FUNCTION_BLOCK AxisMovementController
VAR_INPUT
	tolerance: UINT;
	desiredSpeed: INT;
	currentPosition : UINT;
	requiredPosition : UINT;
END_VAR
VAR_OUTPUT
	AxisMinus : BOOL;
	AxisPlus: BOOL;
	Control: INT;
	SpeedPWM:INT;
	InPosition:BOOL;
END_VAR
VAR
END_VAR

IF  AboutEqual(
	uiActual:= currentPosition,
	uiRequiered:= requiredPosition,
	uiTolerance:= tolerance
)
 THEN
	AxisMinus := FALSE;
	AxisPlus := FALSE;
	Control := 0;
	SpeedPWM := 0;
	InPosition := TRUE;
ELSIF currentPosition > requiredPosition AND NOT InPosition THEN
	AxisMinus := TRUE;
	AxisPlus := FALSE;
	Control:= 32;
	SpeedPWM := desiredSpeed;
	InPosition := FALSE;
ELSIF currentPosition < requiredPosition AND NOT InPosition THEN
	AxisMinus := FALSE;
	AxisPlus := TRUE;
	Control := 32;
	SpeedPWM := desiredSpeed;
	InPosition := FALSE;
ELSE
	AxisMinus := FALSE;
	AxisPlus := FALSE;
	Control := 0;
	SpeedPWM := 0;
	InPosition := FALSE;
END_IF

END_FUNCTION_BLOCK

(* stored: Version 1.1.0.1, ProductVersion 3.1.4024.12
   POU AxisMovementController: Id {02119a59-e7c7-45d5-af1e-b3ec940422ef}, SpecialFunc None *)
